FUNCTION F_Scale : LREAL
VAR_INPUT
	fValue, fMin, fMax	: LREAL;
END_VAR
VAR
	fSpan	: LREAL;
END_VAR

fSpan := fMax - fMin;

IF fSpan = 0 THEN
	F_Scale := 0;
ELSE
	F_Scale := (fValue - fMin) / fSpan;
END_IF

END_FUNCTION

(* stored: Version 1.1.0.1, ProductVersion 3.1.4024.12
   POU F_Scale: Id {9a2bb560-2765-4b4b-b0ec-dc3c3c81d343}, SpecialFunc None *)
